(*
FB indside folder `ExampleFolder`.
*)
FUNCTION_BLOCK FB_ExampleFolder_FunctionBlock

METHOD ExampleFolder_FunctionBlock_Method : BOOL
VAR_INPUT
    input           : BOOL;
END_VAR
END_METHOD

END_FUNCTION_BLOCK

(* stored: Version 1.1.0.1, ProductVersion 3.1.4024.11
   POU FB_ExampleFolder_FunctionBlock: Id {81b96abf-7769-4713-a272-841abc23375b}, SpecialFunc None
   Method ExampleFolder_FunctionBlock_Method: Id {b6c539eb-1440-4463-b6f6-d4f38e958956} *)
